FUNCTION_BLOCK SquareUpMovers EXTENDS FB_DemoStepBase IMPLEMENTS I_TwoMovers
VAR_INPUT
END_VAR
VAR_OUTPUT
END_VAR
VAR
END_VAR

METHOD CyclicLogic
IF Mover.MoveCommand.SquareUp().Done AND Mover2.MoveCommand.SquareUp().Done THEN
			Done:=TRUE;
ELSIF Mover.MoveCommand.SquareUp().Error OR Mover2.MoveCommand.SquareUp().Error THEN
			Step:=E_DemoStep.Disable;
		END_IF
END_METHOD

{error 'Add property implementation or delete property to use base implementation'}
PROPERTY Done : BOOL
GET
END_GET
END_PROPERTY

{warning 'Add property implementation'}
PROPERTY Mover2 : I_XPlanarMover
GET
END_GET
SET
END_SET
END_PROPERTY

END_FUNCTION_BLOCK

(* stored: Version 1.1.0.1, ProductVersion 3.1.4026.19
   POU SquareUpMovers: Id {0243f4e0-eb69-4642-bd5b-6056700c9759}, SpecialFunc None
   Method CyclicLogic: Id {13e63152-bec4-4910-9c94-57f285c6c0e7}
   Property Done: Id {53d7ee30-13ab-4e06-b4c7-e01ebd675f8e}
   Get Get: Id {9c165da7-f5c7-4c05-ba12-f8666675eb7b}
   Property Mover2: Id {ff92c466-7ba1-467d-970d-da1ef653039a}
   Get Get: Id {c3bc423d-4045-4dc6-8a13-aab90e2d79b4}
   Set Set: Id {f59c4d6d-a132-4058-a50d-7b0910799ea3} *)
